FUNCTION_BLOCK CM_ValveWithFB EXTENDS CM_Base IMPLEMENTS I_Valve

VAR_INPUT
	i_stSettings : ST_SettingsValveWithFB;
END_VAR

VAR

	// Inputs
	I_bStaValveIsOn AT %I* : BOOL; //Valve is on (on = positive logic of fuction)
	I_bStaValveIsOff AT %I* : BOOL; //Valve is off
	
	// Outputs
	Q_bCmdOn AT %Q* : BOOL; //Commnad to set valve on
	Q_bCmdOff AT %Q* : BOOL; //Command to set valve off

	// Request
	s_bReqOff : BOOL;
	s_bReqOn : BOOL;
	
	// Status
	s_bStaValveIsOff : BOOL;
	s_bStaValveIsOn : BOOL; 
	
	{attribute: 'Hide'}
	s_bStaValve : BOOL;
	
	{attribute: 'Hide'}
	s_bCfgReverseValve : BOOL; // FALSE = NORMAL, TRUE = INVERTED
	s_bCfgBiStableValve : BOOL; // FALSE = MONO, TRUE = BI
	
	// Alarms
	s_fbAlarmHandlerFeedbackOnTimeout : FB_AlarmHandler;
	s_fbAlarmHandlerFeedbackOffTimeout : FB_AlarmHandler;
	
	s_errFeedbackOnTimeout : BOOL;
	s_errFeedbackOffTimeout : BOOL;
	
	// Timers
	s_tonFeedbackOnTimeout : TON;
	s_tonFeedBackOffTimeout : TON;
END_VAR


SUPER^();

METHOD PROTECTED _m_Alarms : BOOL

IF NOT SUPER^._m_Alarms() THEN
	RETURN;
END_IF

// Timeout (timers)
s_tonFeedBackOffTimeout(
	IN := i_bReqEnable AND s_bReqOff AND NOT(s_bStaValveIsOff),
	PT := i_stSettings.tValveOffTimeout );
	
s_tonFeedbackOnTimeout(
	IN := i_bReqEnable AND s_bReqOn AND NOT(s_bStaValveIsOn),
	PT := i_stSettings.tValveOnTimeout );

// Set error bits
s_errFeedbackOffTimeout := (s_tonFeedBackOffTimeout.Q OR s_errFeedbackOffTimeout) AND NOT(i_bCmdReset);
s_errFeedbackOnTimeout := (s_tonFeedbackOnTimeout.Q OR s_errFeedbackOnTimeout) AND NOT(i_bCmdReset);
	
s_fbAlarmHandlerFeedbackOffTimeout(
	i_bStaActive := i_bReqEnable AND s_errFeedbackOffTimeout, 
	i_eAlarmLevel := E_AlarmLevel.Alarm,
	i_sAlarmText := CONCAT(i_sCmName, ': Feedback off timeout.') );
	
s_fbAlarmHandlerFeedbackOnTimeout(
	i_bStaActive := i_bReqEnable AND s_errFeedbackOnTimeout, 
	i_eAlarmLevel := E_AlarmLevel.Alarm,
	i_sAlarmText := CONCAT(i_sCmName, ': Feedback on timeout.')	);

s_bStaError := 
	s_fbAlarmHandlerFeedbackOffTimeout.q_bStaActive
	OR s_fbAlarmHandlerFeedbackOnTimeout.q_bStaActive;

_m_Alarms := TRUE;
END_METHOD

METHOD PROTECTED _m_Devices : BOOL

IF NOT SUPER^._m_Devices() THEN
	RETURN;
END_IF

_m_Devices := TRUE;
END_METHOD

METHOD PROTECTED _m_Hmi : BOOL

IF NOT SUPER^._m_Hmi() THEN
	RETURN;
END_IF

_m_Hmi := TRUE;
END_METHOD

METHOD PROTECTED _m_Init : BOOL

IF NOT SUPER^._m_Init() THEN
	RETURN;
END_IF

_m_Init := TRUE;
END_METHOD

METHOD PROTECTED _m_Inputs : BOOL

IF NOT SUPER^._m_Inputs() THEN
	RETURN;
END_IF

s_bStaValveIsOff := I_bStaValveIsOff;
s_bStaValveIsOn := I_bStaValveIsOn;

_m_Inputs := TRUE;
END_METHOD

METHOD PROTECTED _m_Outputs : BOOL

IF NOT SUPER^._m_Outputs() THEN
	RETURN;
END_IF

IF s_bCfgBiStableValve THEN
	// BI-STABLE
	Q_bCmdOff := i_bReqEnable AND s_bReqOff AND NOT s_bStaValveIsOff;
	Q_bCmdOn := i_bReqEnable AND s_bReqOn AND NOT s_bStaValveIsOn;
		
ELSE// MONO-STABLE
	IF i_bReqEnable AND s_bReqOff THEN
		Q_bCmdOff := TRUE;
		Q_bCmdOn := FALSE;
	ELSIF i_bReqEnable AND s_bReqOn THEN
		Q_bCmdOff := FALSE;
		Q_bCmdOn := TRUE;
	ELSE
		Q_bCmdOff := FALSE;
		Q_bCmdOn := FALSE;	
	END_IF
	
END_IF
	
_m_Outputs := TRUE;
END_METHOD

METHOD PUBLIC m_Off : BOOL

IF NOT i_bReqEnable THEN 
	RETURN;
END_IF

s_bReqOff := TRUE XOR s_bCfgReverseValve;
s_bReqOn := FALSE XOR s_bCfgReverseValve;

m_Off := TRUE;
END_METHOD

METHOD PUBLIC m_On : BOOL

IF NOT i_bReqEnable THEN 
	RETURN;
END_IF

s_bReqOff := FALSE XOR s_bCfgReverseValve;
s_bReqOn := TRUE XOR s_bCfgReverseValve;

m_On := TRUE;
END_METHOD

METHOD PUBLIC m_Stop : BOOL

IF NOT i_bReqEnable THEN 
	RETURN;
END_IF

s_bReqOff := FALSE;
s_bReqOn := FALSE;

m_Stop := TRUE;
END_METHOD

{attribute 'monitoring':='call'}
PROPERTY PUBLIC p_bCfgBiStableValve : BOOL
GET

p_bCfgBiStableValve := s_bCfgBiStableValve;
END_GET
SET

s_bCfgBiStableValve := p_bCfgBiStableValve;
END_SET
END_PROPERTY

{attribute 'monitoring':='call'}
PROPERTY PUBLIC p_bCfgReverseValve : BOOL
GET

p_bCfgReverseValve := s_bCfgReverseValve;
END_GET
SET

s_bCfgReverseValve := p_bCfgReverseValve;
END_SET
END_PROPERTY

{attribute 'monitoring':='call'}
PROPERTY PUBLIC p_bStaIsOff : BOOL
GET

p_bStaIsOff := s_bStaValveIsOff;
END_GET
END_PROPERTY

{attribute 'monitoring':='call'}
PROPERTY PUBLIC p_bStaIsOn : BOOL
GET

p_bStaIsOn := s_bStaValveIsOn;
END_GET
END_PROPERTY

{attribute 'monitoring':='call'}
PROPERTY PUBLIC p_bStaValve : BOOL
GET

p_bStaValve := s_bStaValveIsOn AND NOT(s_bStaValveIsOff);
END_GET
END_PROPERTY

END_FUNCTION_BLOCK

(* stored: Version 1.1.0.1, ProductVersion 3.1.4024.12
   POU CM_ValveWithFB: Id {4f71df3e-1fa0-4b1d-8b52-9d243bcf380c}, SpecialFunc None
   Folder Methods: Id {ea8d9bb4-734d-4580-8584-865c23a88e42}
   Folder Properties: Id {2ec02995-39e7-4e65-96bd-a76cfe9eceab}
   Method _m_Alarms: Id {d4d0fc1f-8b79-4ff9-9928-983db865f771}
   Method _m_Devices: Id {9853c932-60f5-4fde-8cec-74ce19164cb7}
   Method _m_Hmi: Id {b7e70baf-c92f-407b-8956-5b27f6504914}
   Method _m_Init: Id {aff12dd2-27f0-4c74-8ad8-a313b8d8526f}
   Method _m_Inputs: Id {6569b657-be7e-423b-b5ee-7fd46f745288}
   Method _m_Outputs: Id {96cb9638-dd25-4e5f-a9d1-28835e3be357}
   Method m_Off: Id {dfb0e5fc-71ae-4e37-85af-425dff907aa0}
   Method m_On: Id {7e58f661-0318-4088-96a6-cd17436d0ec9}
   Method m_Stop: Id {c46b72d5-aa2c-476b-88da-c2a403ab692d}
   Property p_bCfgBiStableValve: Id {50a7ecbe-ec5f-4066-8864-d51942ce2c4c}
   Get Get: Id {2aa7ded0-b7cb-4e7f-ac2f-ef302887a57d}
   Set Set: Id {c284b4c5-5788-4a09-a01e-1497eba7f3f7}
   Property p_bCfgReverseValve: Id {897776c2-ad42-4b65-8d5a-3890c3b6823f}
   Get Get: Id {f3fbf4f8-972c-4b1e-966e-d9f0ca7c9f1a}
   Set Set: Id {31b880a5-5c9d-496f-928b-7e6eceda5cde}
   Property p_bStaIsOff: Id {790ca530-7388-4b0e-a36a-513598afadeb}
   Get Get: Id {654072ea-3499-4781-8634-a719128bbe7a}
   Property p_bStaIsOn: Id {f34c7028-14ac-4e6b-8acb-f585d15ae5f6}
   Get Get: Id {1738e38a-8430-47df-b4f9-50a6dbed040c}
   Property p_bStaValve: Id {47f20818-9f3d-497d-8b31-8911fade053e}
   Get Get: Id {95088b72-b64f-4236-9dc6-2cc4fdcc009e} *)
